# EPICS substitutions: iocs/MC06/MCApp/Db-orig/SAI_8MotorStatus.substitutions
file /opt/epics/modules/SAI/db/SAI_8MotorStatus.db {
pattern {	ASYNPORT,	TMOT,		SCAN,		P,		R}
        { 	"pmac",		"1",		".2 second",	"XF:06BM-OP","{Mir:M1}"}
}
